(*********************************** G.D S.p.A. - Technical Department ***********************************
============= PROGRAM INFO ============
FOLDER:             TBD
MACHINES INVOLVED:  TBD 

============= DESCRIPTION =============
csp main interface program

============= REVISIONS ===============
Date		Version	 	Author      	Description             
----------	-------		------------  	--------------------------------------------
2019/09/27 	0000.00	 	M.Grasso		Creation of the PRG

**********************************************************************************************************)
PROGRAM _csp_case_flapControl_highest
VAR
END_VAR

csp_case_flapControl();


		(* LS *)
		(* UPPER *)
			csp_case_fc_ls_upper();
			csp_case_fc_ls_upper_follower();
			csp_case_fc_ls_upper_sensors();
			csp_case_fc_ls_upper_leadingMinorCloser();
			csp_case_fc_ls_upper_leadingMinorCloser_virtual();
			csp_case_fc_ls_upper_spreader();
			(* LOWER *)
			csp_case_fc_ls_lower();
			csp_case_fc_ls_lower_follower();
			csp_case_fc_ls_lower_sensors();
			csp_case_fc_ls_lower_spreader();
			csp_case_fc_ls_lower_trailingCloser();
		(* OS *)
			(* UPPER *)
			csp_case_fc_os_upper();
			csp_case_fc_os_upper_follower();
			csp_case_fc_os_upper_sensors();
			csp_case_fc_os_upper_spreader();
			(* LOWER *)
			csp_case_fc_os_lower();
			csp_case_fc_os_lower_follower();
			csp_case_fc_os_lower_sensors();
			csp_case_fc_os_lower_spreader();

END_PROGRAM

(* stored: Version 1.1.0.1, ProductVersion 3.1.4024.3
   POU _csp_case_flapControl_highest: Id {16373b8f-df73-4324-a592-f49064c802cb}, SpecialFunc None *)
